// Mitsubishi GX Developer project: PLC_PCO520L2   PLC: Q06UDEH

PROGRAM NEW_HMI
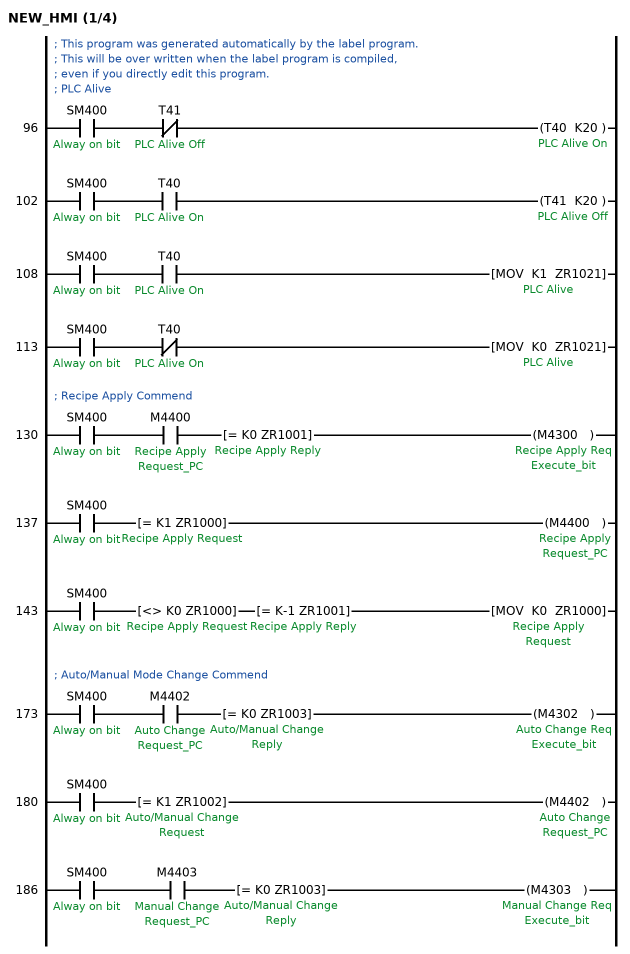
; This program was generated automatically by the label program.
; This will be over written when the label program is compiled,
; even if you directly edit this program.
; PLC Alive
96    LD      SM400  ; Alway on bit
      ANI     T41  ; PLC Alive Off
      OUT     T40 K20  ; PLC Alive On
102   LD      SM400  ; Alway on bit
      AND     T40  ; PLC Alive On
      OUT     T41 K20  ; PLC Alive Off
108   LD      SM400  ; Alway on bit
      AND     T40  ; PLC Alive On
      MOV     K1 ZR1021  ; PLC Alive
113   LD      SM400  ; Alway on bit
      ANI     T40  ; PLC Alive On
      MOV     K0 ZR1021
; Recipe Apply Commend
130   LD      SM400  ; Alway on bit
      AND     M4400  ; Recipe Apply Request_PC
      AND=    K0 ZR1001  ; Recipe Apply Reply
      OUT     M4300  ; Recipe Apply Req Execute_bit
137   LD      SM400  ; Alway on bit
      AND=    K1 ZR1000  ; Recipe Apply Request
      OUT     M4400  ; Recipe Apply Request_PC
143   LD      SM400  ; Alway on bit
      AND<>   K0 ZR1000  ; Recipe Apply Request
      AND=    K-1 ZR1001  ; Recipe Apply Reply
      MOV     K0 ZR1000
; Auto/Manual Mode Change Commend
173   LD      SM400  ; Alway on bit
      AND     M4402  ; Auto Change Request_PC
      AND=    K0 ZR1003  ; Auto/Manual Change Reply
      OUT     M4302  ; Auto Change Req Execute_bit
180   LD      SM400  ; Alway on bit
      AND=    K1 ZR1002  ; Auto/Manual Change Request
      OUT     M4402  ; Auto Change Request_PC
186   LD      SM400  ; Alway on bit
      AND     M4403  ; Manual Change Request_PC
      AND=    K0 ZR1003  ; Auto/Manual Change Reply
      OUT     M4303  ; Manual Change Req Execute_bit
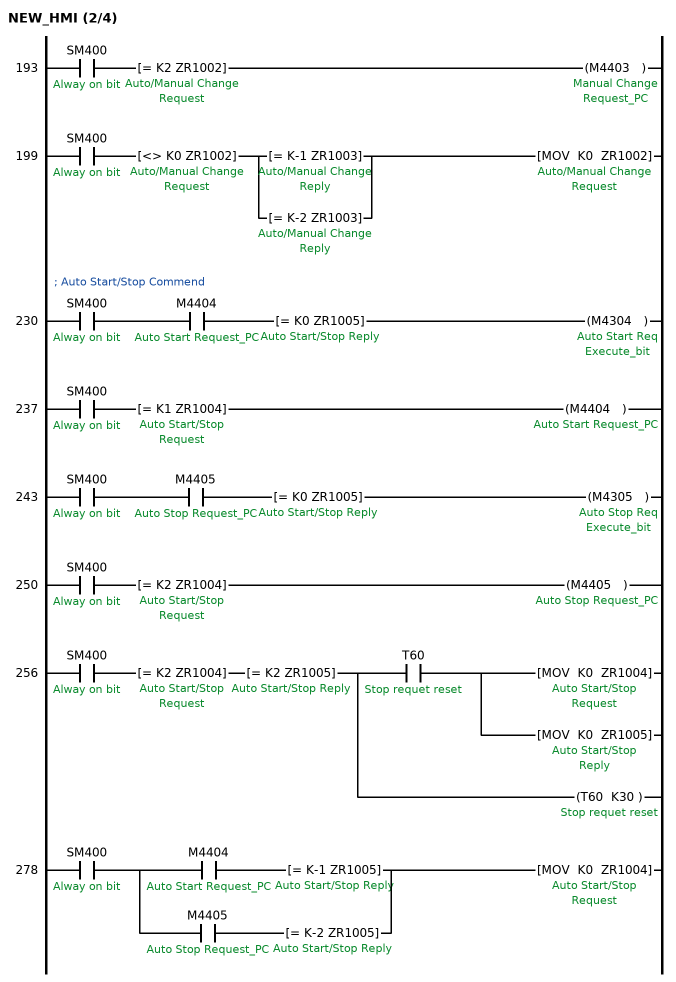
193   LD      SM400  ; Alway on bit
      AND=    K2 ZR1002  ; Auto/Manual Change Request
      OUT     M4403  ; Manual Change Request_PC
199   LD      SM400  ; Alway on bit
      AND<>   K0 ZR1002  ; Auto/Manual Change Request
      LD=     K-1 ZR1003  ; Auto/Manual Change Reply
      OR=     K-2 ZR1003  ; Auto/Manual Change Reply
      ANB
      MOV     K0 ZR1002
; Auto Start/Stop Commend
230   LD      SM400  ; Alway on bit
      AND     M4404  ; Auto Start Request_PC
      AND=    K0 ZR1005  ; Auto Start/Stop Reply
      OUT     M4304  ; Auto Start Req Execute_bit
237   LD      SM400  ; Alway on bit
      AND=    K1 ZR1004  ; Auto Start/Stop Request
      OUT     M4404  ; Auto Start Request_PC
243   LD      SM400  ; Alway on bit
      AND     M4405  ; Auto Stop Request_PC
      AND=    K0 ZR1005  ; Auto Start/Stop Reply
      OUT     M4305  ; Auto Stop Req Execute_bit
250   LD      SM400  ; Alway on bit
      AND=    K2 ZR1004  ; Auto Start/Stop Request
      OUT     M4405  ; Auto Stop Request_PC
256   LD      SM400  ; Alway on bit
      AND=    K2 ZR1004  ; Auto Start/Stop Request
      AND=    K2 ZR1005  ; Auto Start/Stop Reply
      MPS
      AND     T60  ; Stop requet reset
      MOV     K0 ZR1004
      MOV     K0 ZR1005
      MPP
      OUT     T60 K30  ; Stop requet reset
278   LD      SM400  ; Alway on bit
      LD      M4404  ; Auto Start Request_PC
      AND=    K-1 ZR1005  ; Auto Start/Stop Reply
      LD      M4405  ; Auto Stop Request_PC
      AND=    K-2 ZR1005  ; Auto Start/Stop Reply
      ORB
      ANB
      MOV     K0 ZR1004
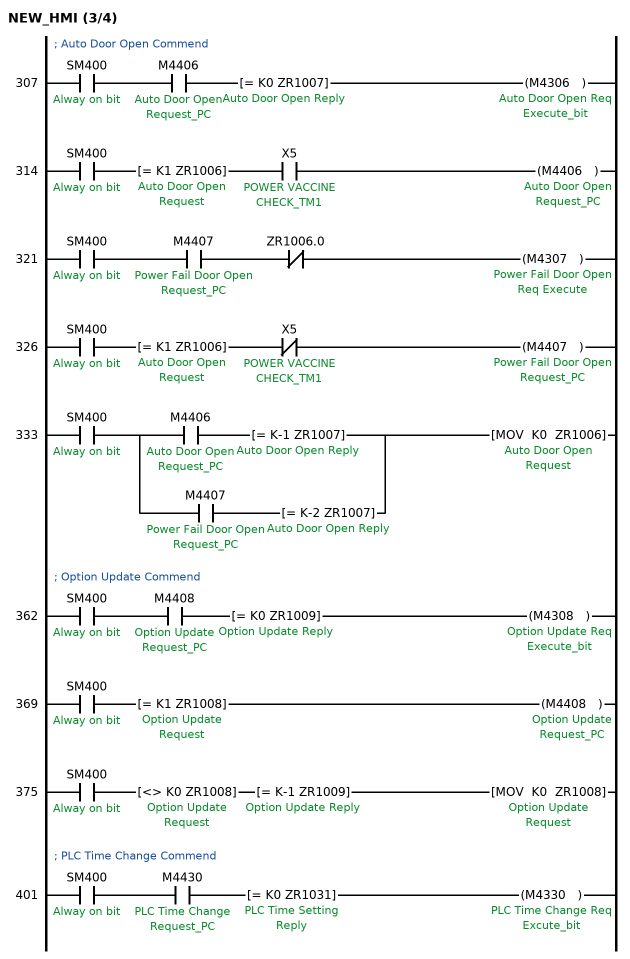
; Auto Door Open Commend
307   LD      SM400  ; Alway on bit
      AND     M4406  ; Auto Door Open Request_PC
      AND=    K0 ZR1007  ; Auto Door Open Reply
      OUT     M4306  ; Auto Door Open Req Execute_bit
314   LD      SM400  ; Alway on bit
      AND=    K1 ZR1006  ; Auto Door Open Request
      AND     X5  ; POWER VACCINE CHECK_TM1
      OUT     M4406  ; Auto Door Open Request_PC
321   LD      SM400  ; Alway on bit
      AND     M4407  ; Power Fail Door Open Request_PC
      ANI     ZR1006.0
      OUT     M4307  ; Power Fail Door Open Req Execute
326   LD      SM400  ; Alway on bit
      AND=    K1 ZR1006  ; Auto Door Open Request
      ANI     X5  ; POWER VACCINE CHECK_TM1
      OUT     M4407  ; Power Fail Door Open Request_PC
333   LD      SM400  ; Alway on bit
      LD      M4406  ; Auto Door Open Request_PC
      AND=    K-1 ZR1007  ; Auto Door Open Reply
      LD      M4407  ; Power Fail Door Open Request_PC
      AND=    K-2 ZR1007  ; Auto Door Open Reply
      ORB
      ANB
      MOV     K0 ZR1006
; Option Update Commend
362   LD      SM400  ; Alway on bit
      AND     M4408  ; Option Update Request_PC
      AND=    K0 ZR1009  ; Option Update Reply
      OUT     M4308  ; Option Update Req Execute_bit
369   LD      SM400  ; Alway on bit
      AND=    K1 ZR1008  ; Option Update Request
      OUT     M4408  ; Option Update Request_PC
375   LD      SM400  ; Alway on bit
      AND<>   K0 ZR1008  ; Option Update Request
      AND=    K-1 ZR1009  ; Option Update Reply
      MOV     K0 ZR1008
; PLC Time Change Commend
401   LD      SM400  ; Alway on bit
      AND     M4430  ; PLC Time Change Request_PC
      AND=    K0 ZR1031  ; PLC Time Setting Reply
      OUT     M4330  ; PLC Time Change Req Excute_bit
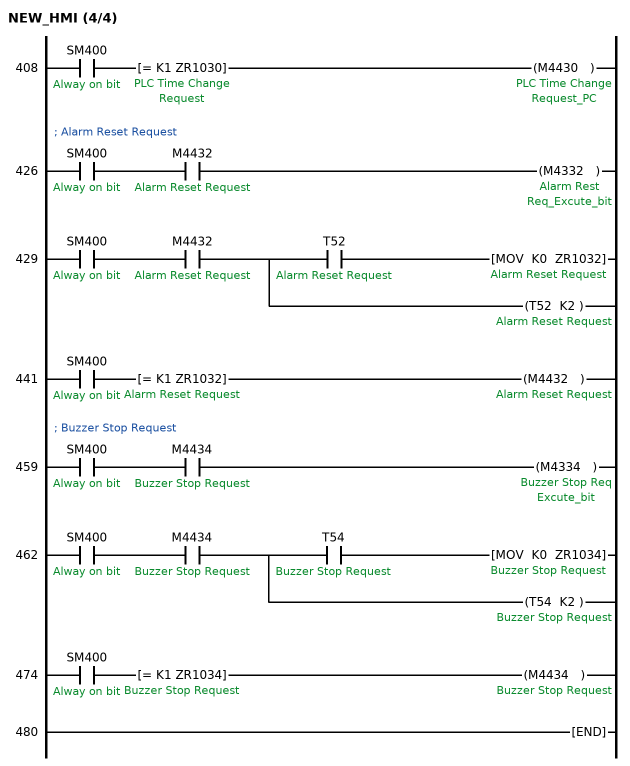
408   LD      SM400  ; Alway on bit
      AND=    K1 ZR1030  ; PLC Time Change Request
      OUT     M4430  ; PLC Time Change Request_PC
; Alarm Reset Request
426   LD      SM400  ; Alway on bit
      AND     M4432  ; Alarm Reset Request
      OUT     M4332  ; Alarm Rest Req_Excute_bit
429   LD      SM400  ; Alway on bit
      AND     M4432  ; Alarm Reset Request
      MPS
      AND     T52  ; Alarm Reset Request
      MOV     K0 ZR1032  ; Alarm Reset Request
      MPP
      OUT     T52 K2  ; Alarm Reset Request
441   LD      SM400  ; Alway on bit
      AND=    K1 ZR1032  ; Alarm Reset Request
      OUT     M4432  ; Alarm Reset Request
; Buzzer Stop Request
459   LD      SM400  ; Alway on bit
      AND     M4434  ; Buzzer Stop Request
      OUT     M4334  ; Buzzer Stop Req Excute_bit
462   LD      SM400  ; Alway on bit
      AND     M4434  ; Buzzer Stop Request
      MPS
      AND     T54  ; Buzzer Stop Request
      MOV     K0 ZR1034  ; Buzzer Stop Request
      MPP
      OUT     T54 K2  ; Buzzer Stop Request
474   LD      SM400  ; Alway on bit
      AND=    K1 ZR1034  ; Buzzer Stop Request
      OUT     M4434  ; Buzzer Stop Request
480   END
END_PROGRAM
